// TwinCAT 3 PLC project TcAlarms
// Title: TwinCAT Alarm Handling Library
// Company: https://github.com/petr-suchy
// Author: Petr Suchý
// ProjectVersion: 0.0.1.0
// Description: TwinCAT library for alarm handling in PLC programs.
// ProgramVersion: 3.1.4024.0
// libraries:
//   Tc2_Standard, * (Beckhoff Automation GmbH)
//   Tc2_System, * (Beckhoff Automation GmbH)
//   Tc3_Module, * (Beckhoff Automation GmbH)
// project tree:
//   Alarms/DUTs/ E_AlarmSeverity.TcDUT, E_ArgType.TcDUT, ST_AlarmElement.TcDUT (not stored), ST_AlarmPageRow.TcDUT (not stored), ST_Arg.TcDUT (not stored)
//   Alarms/FBs/ FB_Alarm.TcPOU, FB_AlarmArg.TcPOU (not stored), FB_AlarmBase.TcPOU, FB_AlarmContext.TcPOU, FB_ArgStack.TcPOU, FB_RdArgStack.TcPOU, FB_SRAlarm.TcPOU (not stored), FB_SRAlarmArg.TcPOU, FB_VFormatStr.TcPOU, FB_WrArgStack.TcPOU
//   Alarms/FUNs/ A_BOOL.TcPOU (not stored), A_BYTE.TcPOU (not stored), A_DATE.TcPOU, A_DINT.TcPOU (not stored), A_DWORD.TcPOU (not stored), A_INT.TcPOU, A_LREAL.TcPOU (not stored), A_REAL.TcPOU, A_SINT.TcPOU (not stored), A_STRING.TcPOU (not stored), A_TIME.TcPOU, A_UDINT.TcPOU (not stored), A_UINT.TcPOU, A_USINT.TcPOU, A_WORD.TcPOU
//   Alarms/GVLs/ GVL_Alarms.TcGVL
//   Alarms/ITFs/ I_Alarm.TcIO, I_AlarmContext.TcIO, I_AlarmTextList.TcIO (not stored)
//   / ImagePool_Alarms.TcIPO (not stored), PlcTask.TcTTO
//   Memory/DUTs/ ST_SIZE.TcDUT
//   Memory/FUNs/ WORD_TO_SIZE.TcPOU, DINT_TO_SIZE.TcPOU, INT_TO_SIZE.TcPOU, F_MemCpy.TcPOU, F_MemSet.TcPOU, SINT_TO_SIZE.TcPOU, SIZE_TO_VALUE.TcPOU, UDINT_TO_SIZE.TcPOU, UINT_TO_SIZE.TcPOU, USINT_TO_SIZE.TcPOU, BYTE_TO_SIZE.TcPOU, DWORD_TO_SIZE.TcPOU
//   POUs/ MAIN.TcPOU
//   Version/ Global_Version.TcGVL
// real-time tasks:
//   TASK PlcTask: cycle T#10ms, priority 20, ADS port 350

CONFIGURATION TcAlarms
    RESOURCE PLC ON TwinCAT3
        TASK PlcTask(INTERVAL := T#10ms, PRIORITY := 20);
        PROGRAM MAIN WITH PlcTask : MAIN;
    END_RESOURCE
END_CONFIGURATION

// ---- Alarms/DUTs/E_AlarmSeverity.TcDUT
{attribute 'qualified_only'}
{attribute 'strict'}
{attribute 'to_string'}
TYPE E_AlarmSeverity :
(
	NoneAlarm := 0,
	InfoAlarm,
	WarningAlarm,
	ErrorAlarm
) BYTE := NoneAlarm;
END_TYPE

// ---- Alarms/DUTs/E_ArgType.TcDUT
{attribute 'qualified_only'}
{attribute 'strict'}
TYPE E_ArgType :
(
	VoidArg := 0,
	BoolArg,
	ByteArg,
	WordArg,
	DWordArg,
	SIntArg,
	USIntArg,
	IntArg,
	UIntArg,
	DIntArg,
	UDIntArg,
	RealArg,
	LRealArg,
	StringArg,
	TimeArg,
	DateArg
) BYTE := VoidArg;
END_TYPE

// ---- Memory/DUTs/ST_SIZE.TcDUT
TYPE ST_SIZE :
STRUCT
	nValue : UDINT;
END_STRUCT
END_TYPE

// ---- Alarms/GVLs/GVL_Alarms.TcGVL
VAR_GLOBAL CONSTANT
	ALARM_INVALID_CONTEXT_ID	: DINT := 0;
	ALARM_INVALID_INDEX			: DINT := -1;
	ALARM_ARG_STACK_SIZE		: DINT := 255;
	ALARM_TEXT_SIZE				: INT := 255;
END_VAR

// ---- Version/Global_Version.TcGVL
{attribute 'TcGenerated'}
{attribute 'no-analysis'}
{attribute 'linkalways'}
// This function has been automatically generated from the project information.
VAR_GLOBAL CONSTANT
	{attribute 'const_non_replaced'}
	stLibVersion_TwinCAT_Alarm_Handling_Library : ST_LibVersion := (iMajor := 0, iMinor := 0, iBuild := 1, iRevision := 0, nFlags := 0, sVersion := '0.0.1.0');
END_VAR

// ---- Alarms/ITFs/I_Alarm.TcIO
INTERFACE I_Alarm

PROPERTY AlarmId : DINT
GET
END_GET
END_PROPERTY

PROPERTY AlarmSeverity : E_AlarmSeverity
GET
END_GET
END_PROPERTY

PROPERTY ArgStackMemoryPointer : POINTER TO BYTE
GET
END_GET
END_PROPERTY

PROPERTY ArgStackMemorySize : DINT
GET
END_GET
END_PROPERTY

END_INTERFACE

// ---- Alarms/ITFs/I_AlarmContext.TcIO
INTERFACE I_AlarmContext

PROPERTY Acknowledge : BOOL
GET
END_GET
END_PROPERTY

METHOD AddNewAlarm : DINT
VAR_INPUT
	iAlarm : I_Alarm;
END_VAR
END_METHOD

METHOD EnableAcknowledge : BOOL
VAR_INPUT
	nAlarmContextId		: DINT;
	bCanByAcknowledged	: BOOL;
END_VAR
END_METHOD

PROPERTY IsAlarmBufferFull : BOOL
GET
END_GET
END_PROPERTY

METHOD RemoveAlarm : BOOL
VAR_INPUT
	nAlarmContextId : DINT;
END_VAR
END_METHOD

PROPERTY SelectedAlarmContextId : DINT
GET
END_GET
END_PROPERTY

END_INTERFACE

// ---- POUs/MAIN.TcPOU
PROGRAM MAIN
VAR
END_VAR

END_PROGRAM

// ---- Alarms/FBs/FB_Alarm.TcPOU
FUNCTION_BLOCK FB_Alarm EXTENDS FB_AlarmBase
VAR_INPUT
	bEnable				: BOOL;
END_VAR

bActive := bEnable;

SUPER^();

PROPERTY ArgStackMemoryPointer : POINTER TO BYTE
GET
ArgStackMemoryPointer := 0;
END_GET
END_PROPERTY

PROPERTY ArgStackMemorySize : DINT
GET
ArgStackMemorySize := 0;
END_GET
END_PROPERTY

METHOD PROTECTED  ClearArgStack
VAR_INPUT
END_VAR
// Do nothing
END_METHOD

METHOD PROTECTED CopyArgsToStack
VAR_INPUT
END_VAR
// Do nothing
END_METHOD

END_FUNCTION_BLOCK

// ---- Alarms/FBs/FB_AlarmBase.TcPOU
FUNCTION_BLOCK ABSTRACT FB_AlarmBase IMPLEMENTS I_Alarm
VAR_OUTPUT
	bActive				: BOOL;
END_VAR
VAR
	iAlarmContext		: I_AlarmContext;
	nAlarmContextId		: DINT := ALARM_INVALID_CONTEXT_ID;
	eAlarmSeverity		: E_AlarmSeverity;
	nAlarmId			: DINT;
	fbActiveRTrig		: R_TRIG;
	fbActiveFTrig		: F_TRIG;
END_VAR

fbActiveRTrig(CLK := bActive);
fbActiveFTrig(CLK := bActive);

IF fbActiveRTrig.Q THEN
	CopyArgsToStack();
END_IF

IF bActive AND nAlarmContextId = ALARM_INVALID_CONTEXT_ID AND NOT iAlarmContext.IsAlarmBufferFull THEN
	// Add this alarm to alarm context
	nAlarmContextId := iAlarmContext.AddNewAlarm(THIS^);
END_IF

IF fbActiveFTrig.Q THEN
	IF nAlarmContextId <> ALARM_INVALID_CONTEXT_ID THEN
		// Prepare argument stack for new arguments
		ClearArgStack();
		// Remove this alarm from alarm context
		iAlarmContext.RemoveAlarm(nAlarmContextId);
		nAlarmContextId := ALARM_INVALID_CONTEXT_ID;
	END_IF
END_IF

PROPERTY AlarmId : DINT
GET
AlarmId := nAlarmId;
END_GET
END_PROPERTY

PROPERTY AlarmSeverity : E_AlarmSeverity
GET
AlarmSeverity := eAlarmSeverity;
END_GET
END_PROPERTY

PROPERTY ABSTRACT ArgStackMemoryPointer : POINTER TO BYTE
GET
END_GET
END_PROPERTY

PROPERTY ABSTRACT ArgStackMemorySize : DINT
GET
END_GET
END_PROPERTY

METHOD PROTECTED ABSTRACT ClearArgStack
VAR_INPUT
END_VAR
END_METHOD

METHOD PROTECTED ABSTRACT CopyArgsToStack
VAR_INPUT
END_VAR
END_METHOD

METHOD FB_init : BOOL
VAR_INPUT
	bInitRetains		: BOOL; // if TRUE, the retain variables are initialized (warm start / cold start)
	bInCopyCode			: BOOL;  // if TRUE, the instance afterwards gets moved into the copy code (online change)
	iAlarmContext		: I_AlarmContext;
	eAlarmSeverity		: E_AlarmSeverity;
	nAlarmId			: DINT;
END_VAR
THIS^.iAlarmContext := iAlarmContext;
THIS^.eAlarmSeverity := eAlarmSeverity;
THIS^.nAlarmId := nAlarmId;
END_METHOD

END_FUNCTION_BLOCK

// ---- Alarms/FBs/FB_AlarmContext.TcPOU
FUNCTION_BLOCK FB_AlarmContext IMPLEMENTS I_AlarmContext
VAR_INPUT
	bEnable						: BOOL;
	bFirstAlarm					: BOOL;
	bLastAlarm					: BOOL;
	bPrevAlarm					: BOOL;
	bNextAlarm					: BOOL;
	bAcknowledge				: BOOL;
END_VAR
VAR_OUTPUT
	bActive						: BOOL;
	nNumOfDisplayedAlarms		: DINT;
END_VAR
VAR_IN_OUT
	aAlarmPage					: ARRAY[*] OF ST_AlarmPageRow;
	nSelectedAlarm				: INT;
END_VAR
VAR
	pAlarmArray					: POINTER TO ST_AlarmElement;
	nMaxNumOfAlarms				: DINT;
	iAlarmTextList				: I_AlarmTextList;
	nNumOfAlarms				: DINT;
	nNextContextId				: DINT := ALARM_INVALID_CONTEXT_ID + 1;
	nSelectedAlarmContextId		: DINT := ALARM_INVALID_CONTEXT_ID;
	fbEnableFTrig				: F_TRIG;
	fbFirstAlarmRTrig			: R_TRIG;
	fbLastAlarmRTrig			: R_TRIG;
	fbPrevAlarmRTrig			: R_TRIG;
	fbNextAlarmRTrig			: R_TRIG;
	fbVFormatStr				: FB_VFormatStr;
	// Index of the first alarm in the alarm array to be displayed
	nFirstAlarmToDisplay		: DINT;
	// Number of alarm selected in table
	nSelectedAlarm_				: DINT;
END_VAR
VAR_TEMP
	nPageLBound					: DINT;
	nPageUBound					: DINT;
	nPageSize					: DINT;
	nActualNumOfAlarms			: DINT;
	nSelectedAlarmOffset		: DINT;
	stCurrAlarm					: REFERENCE TO ST_AlarmElement;
	stCurrPageRow				: REFERENCE TO ST_AlarmPageRow;
	i							: DINT;
END_VAR

bActive := bEnable;
nSelectedAlarmContextId := ALARM_INVALID_CONTEXT_ID;

fbEnableFTrig(CLK := bEnable);

fbFirstAlarmRTrig(CLK := bFirstAlarm);
fbLastAlarmRTrig(CLK := bLastAlarm);
fbPrevAlarmRTrig(CLK := bPrevAlarm);
fbNextAlarmRTrig(CLK := bNextAlarm);

// The first index in the output array
nPageLBound := LOWER_BOUND(aAlarmPage, 1);
// The last index in the output array
nPageUBound := UPPER_BOUND(aAlarmPage, 1);
// Size of the output array
nPageSize := nPageUBound - nPageLBound + 1;

IF fbEnableFTrig.Q THEN
	// Reset FB output when enable is lost
	FOR i := nPageLBound TO nPageUBound DO
		ClearPageRow(i);
	END_FOR
	nNumOfDisplayedAlarms := 0;
END_IF

IF NOT bEnable THEN
	RETURN;
END_IF

// Get alarm number from FB input
nSelectedAlarm_ := nSelectedAlarm;

// Restrict index to the lower limit
nSelectedAlarm_ := MAX(nPageLBound, nSelectedAlarm_);
// Restrict index to the upper limit
nSelectedAlarm_ := MIN(nPageUBound, nSelectedAlarm_);

// Go to the first alarm
IF fbFirstAlarmRTrig.Q THEN
	nFirstAlarmToDisplay := 0;
	nSelectedAlarm_ := nPageLBound;
END_IF

// Go to the last alarm
IF fbLastAlarmRTrig.Q THEN
	nFirstAlarmToDisplay := (nNumOfAlarms / nPageSize) * nPageSize;
	nSelectedAlarm_ := MAX(nNumOfAlarms MOD nPageSize, 1);
END_IF

// Go to the previous alarm
IF fbPrevAlarmRTrig.Q THEN
	// Is the first alarm on the alarm page selected?
	IF nSelectedAlarm_ <= nPageLBound THEN
		// Move displayed alarms backward by one
		nFirstAlarmToDisplay := nFirstAlarmToDisplay - 1;
	ELSE
		// Select previous alarm
		nSelectedAlarm_ := nSelectedAlarm_ - 1;
	END_IF
END_IF

// Go to the next alarm
IF fbNextAlarmRTrig.Q THEN
	// Is the last alarm on the alarm page selected?
	IF nSelectedAlarm_ >= nPageUBound THEN
		IF nNumOfAlarms > nPageSize THEN
			// Move displayed alarms forward by one
			nFirstAlarmToDisplay := nFirstAlarmToDisplay + 1;
		END_IF
	ELSE
		// Select next alarm
		nSelectedAlarm_ := nSelectedAlarm_ + 1;
	END_IF
END_IF

// Return selected alarm back to the FB output
nSelectedAlarm := DINT_TO_INT(nSelectedAlarm_);

// Restrict alarm index to the upper limit
nFirstAlarmToDisplay := MIN(nFirstAlarmToDisplay, nNumOfAlarms - 1);
// Restrict alarm index to the lower limit
nFirstAlarmToDisplay := MAX(nFirstAlarmToDisplay, 0);

// Actual number of alarms that can be displayed
nActualNumOfAlarms := nNumOfAlarms - nFirstAlarmToDisplay;
// Number of alarms to be displayed
nNumOfDisplayedAlarms := MIN(nPageSize, nActualNumOfAlarms);

FOR i := 0 TO nNumOfDisplayedAlarms - 1 DO
	
	stCurrAlarm REF= pAlarmArray[nFirstAlarmToDisplay + i];
	stCurrPageRow REF= aAlarmPage[nPageLBound + i];

	// Convert alarm severity to string
	stCurrPageRow.sAlarmSeverity := TO_STRING(stCurrAlarm.eAlarmSeverity);
	// Convert alarm id to string
	stCurrPageRow.sAlarmId := DINT_TO_STRING(stCurrAlarm.nAlarmId);	
	// Format alarm text using the argument stack
	fbVFormatStr(
		sFormat := iAlarmTextList.GetAlarmText(stCurrAlarm.nAlarmId),
		pArgStack := ADR(stCurrAlarm.aArgStack), 
		nStackSize := SIZEOF(stCurrAlarm.aArgStack),
		sOutput => stCurrPageRow.sAlarmText
	);
	// Convert Ack flag to string
	IF stCurrAlarm.bCanByAcknowledged THEN
		stCurrPageRow.sCanByAcknowledged := '!';
	ELSE
		stCurrPageRow.sCanByAcknowledged := '';
	END_IF
END_FOR

// Clear the rest of the output array
FOR i := nPageLBound + nNumOfDisplayedAlarms TO nPageUBound DO
	ClearPageRow(i);
END_FOR

// Get context id of selected alarm
IF nPageLBound <= nSelectedAlarm_ AND nSelectedAlarm_ <= nPageUBound THEN
	nSelectedAlarmOffset := nSelectedAlarm_ - nPageLBound;
	IF nSelectedAlarmOffset < nNumOfDisplayedAlarms THEN
		nSelectedAlarmContextId := pAlarmArray[nFirstAlarmToDisplay + nSelectedAlarmOffset].nAlarmContextId;
	END_IF
END_IF

PROPERTY Acknowledge : BOOL
GET
Acknowledge := bAcknowledge;
END_GET
END_PROPERTY

METHOD PUBLIC AddNewAlarm : DINT
VAR_INPUT
	iAlarm : I_Alarm;
END_VAR
VAR
	i : DINT;
END_VAR
AddNewAlarm := ALARM_INVALID_CONTEXT_ID;

IF NOT IsAlarmBufferFull THEN

	// Make space for a new alarm by shifting array elements to right
	FOR i := 1 TO nNumOfAlarms DO
		pAlarmArray[nNumOfAlarms - i + 1] := pAlarmArray[nNumOfAlarms - i];
	END_FOR
	
	pAlarmArray[0].nAlarmContextId := nNextContextId;
	pAlarmArray[0].eAlarmSeverity := iAlarm.AlarmSeverity; 
	pAlarmArray[0].nAlarmId := iAlarm.AlarmId;
	pAlarmArray[0].bCanByAcknowledged := FALSE;
	
	IF iAlarm.ArgStackMemoryPointer <> 0 AND iAlarm.ArgStackMemorySize > 0 THEN
		F_MemCpy(
			pDestAddr:= ADR(pAlarmArray[0].aArgStack),
			stDestSize:= UDINT_TO_SIZE(SIZEOF(pAlarmArray[0].aArgStack)),
			pSrcAddr:= iAlarm.ArgStackMemoryPointer,
			stSrcSize:= DINT_TO_SIZE(iAlarm.ArgStackMemorySize));
	END_IF

	nNextContextId := nNextContextId + 1;
	
	// Prevent context id overflow
	IF nNextContextId <= ALARM_INVALID_CONTEXT_ID THEN
		nNextContextId := ALARM_INVALID_CONTEXT_ID + 1;
	END_IF
	
	nNumOfAlarms := nNumOfAlarms + 1;

	AddNewAlarm := pAlarmArray[0].nAlarmContextId;
END_IF
END_METHOD

METHOD PRIVATE ClearPageRow
VAR_INPUT
	nRowIdx : DINT;
END_VAR
aAlarmPage[nRowIdx].sAlarmSeverity := TO_STRING(E_AlarmSeverity.NoneAlarm);
aAlarmPage[nRowIdx].sAlarmId := '';
aAlarmPage[nRowIdx].sAlarmText := '';
aAlarmPage[nRowIdx].sCanByAcknowledged := '';
END_METHOD

METHOD PUBLIC EnableAcknowledge : BOOL
VAR_INPUT
	nAlarmContextId		: DINT;
	bCanByAcknowledged	: BOOL;
END_VAR
VAR
	nArrayIndex			: DINT;
END_VAR
EnableAcknowledge := FALSE;
nArrayIndex := GetArrayIndexByContextId(nAlarmContextId);

IF nArrayIndex <> ALARM_INVALID_INDEX THEN
	pAlarmArray[nArrayIndex].bCanByAcknowledged := bCanByAcknowledged;
	EnableAcknowledge := TRUE;
END_IF
END_METHOD

METHOD FB_init : BOOL
VAR_INPUT
	bInitRetains			: BOOL;								// if TRUE, the retain variables are initialized (warm start / cold start)
	bInCopyCode				: BOOL;								// if TRUE, the instance afterwards gets moved into the copy code (online change)
	pAlarmArray				: POINTER TO ST_AlarmElement;
	nMaxNumOfAlarms			: DINT;
	iAlarmTextList			: I_AlarmTextList;
END_VAR
THIS^.pAlarmArray := pAlarmArray;
THIS^.nMaxNumOfAlarms := nMaxNumOfAlarms;
THIS^.iAlarmTextList := iAlarmTextList;
END_METHOD

METHOD PRIVATE GetArrayIndexByContextId : DINT
VAR_INPUT
	nAlarmContextId : DINT;
END_VAR
VAR
	i : DINT;
END_VAR
GetArrayIndexByContextId := ALARM_INVALID_INDEX;

IF nAlarmContextId <> ALARM_INVALID_CONTEXT_ID THEN
	FOR i := 0 TO nNumOfAlarms - 1 DO
		IF pAlarmArray[i].nAlarmContextId = nAlarmContextId THEN
			GetArrayIndexByContextId := i;
			RETURN;
		END_IF
	END_FOR
END_IF
END_METHOD

PROPERTY PUBLIC IsAlarmBufferFull : BOOL
GET
IsAlarmBufferFull := nNumOfAlarms >= nMaxNumOfAlarms;
END_GET
END_PROPERTY

METHOD PUBLIC RemoveAlarm : BOOL
VAR_INPUT
	nAlarmContextId		: DINT;
END_VAR
VAR
	nArrayIndex			: DINT;
	i					: DINT;
END_VAR
RemoveAlarm := FALSE;
nArrayIndex := GetArrayIndexByContextId(nAlarmContextId);

IF nArrayIndex > ALARM_INVALID_INDEX AND nArrayIndex < nNumOfAlarms THEN

	// Remove element from array by shifting array elements to left
	FOR i := nArrayIndex TO nNumOfAlarms - 2 DO
		pAlarmArray[i] := pAlarmArray[i + 1];
	END_FOR
	nNumOfAlarms := nNumOfAlarms - 1;
	
	// Reinitialise element at the end of array freed by shifting
	pAlarmArray[nNumOfAlarms].nAlarmContextId := ALARM_INVALID_CONTEXT_ID;
	pAlarmArray[nNumOfAlarms].nAlarmId := 0;
	pAlarmArray[nNumOfAlarms].bCanByAcknowledged := FALSE;
	
	F_MemSet(
		pDestAddr:= ADR(pAlarmArray[nNumOfAlarms].aArgStack),
		nWithChar:= 0,
		stDestSize:= UDINT_TO_SIZE(SIZEOF(pAlarmArray[nNumOfAlarms].aArgStack)));

	RemoveAlarm := TRUE;
END_IF
END_METHOD

PROPERTY PUBLIC SelectedAlarmContextId : DINT
GET
SelectedAlarmContextId := nSelectedAlarmContextId;
END_GET
END_PROPERTY

END_FUNCTION_BLOCK

// ---- Alarms/FBs/FB_VFormatStr.TcPOU
FUNCTION_BLOCK FB_VFormatStr
VAR_INPUT
	sFormat			: STRING(ALARM_TEXT_SIZE);
	pArgStack		: POINTER TO BYTE;
	nStackSize		: DINT;
END_VAR
VAR_OUTPUT
	sOutput			: STRING(ALARM_TEXT_SIZE);
END_VAR
VAR
	fbRdArgStack		: FB_RdArgStack(0, 0);
	nFormatLength		: INT;
	nCurrFormatIndex	: INT;
	nCurrOutputIndex	: INT;
	i					: INT;
	c					: BYTE;
END_VAR
VAR CONSTANT
	SPEC_CHAR	: BYTE := 37;	// '%'
	SPEC_D		: BYTE := 100;	// '%d'
	SPEC_F		: BYTE := 102;	// '%f'
	SPEC_S		: BYTE := 115;	// '%s'
	SPEC_TIME	: BYTE := 84;	// %T
	SPEC_DATE	: BYTE := 68;	// %D
END_VAR

fbRdArgStack.SetMemory(pArgStack, nStackSize);

// Zero output string
F_MemSet(
	pDestAddr:= ADR(sOutput),
	nWithChar:= 0,
	stDestSize:= UDINT_TO_SIZE(SIZEOF(sOutput)));

// Get format string length
nFormatLength := LEN(sFormat);

nCurrFormatIndex := 0;
nCurrOutputIndex := 0;

WHILE NOT AtFmtEnd DO
	
	c := FmtChar;
	NextFmtChar();
	
	IF c = SPEC_CHAR THEN
		
		IF AtFmtEnd THEN
			PutChar(c);
			EXIT;
		END_IF
		
		c := FmtChar;
		NextFmtChar();
	
		CASE c OF
			SPEC_D:
				IF fbRdArgStack.IsIntArg THEN
					PutStr(DINT_TO_STRING(fbRdArgStack.GetIntArg()));
				ELSIF fbRdArgStack.IsUIntArg THEN
					PutStr(UDINT_TO_STRING(fbRdArgStack.GetUIntArg()));
				ELSE
					PutStr('???');
				END_IF
				fbRdArgStack.NextArg();
			SPEC_F:
				IF fbRdArgStack.IsFloatArg THEN
					PutStr(LREAL_TO_STRING(fbRdArgStack.GetFloatArg()));
				ELSE
					PutStr('???');
				END_IF
				fbRdArgStack.NextArg();
			SPEC_S:
				IF fbRdArgStack.IsString THEN
					PutStr(fbRdArgStack.GetStringArg());
				ELSE
					PutStr('???');
				END_IF
			SPEC_TIME:
				IF fbRdArgStack.IsTime THEN
					PutStr(TIME_TO_STRING(fbRdArgStack.GetTimeArg()));
				ELSE
					PutStr('???');
				END_IF
			SPEC_DATE:
				IF fbRdArgStack.IsDate THEN
					PutStr(DATE_TO_STRING(fbRdArgStack.GetDateArg()));
				ELSE
					PutStr('???');
				END_IF			
		ELSE
			IF c = SPEC_CHAR THEN // %% escape sequence?
				PutChar(c);
			ELSE
				PutChar(SPEC_CHAR);
				PutChar(c);
			END_IF
		END_CASE
	ELSE
		PutChar(c);
	END_IF
END_WHILE

PROPERTY PRIVATE AtFmtEnd : BOOL
GET
AtFmtEnd := nCurrFormatIndex >= nFormatLength;
END_GET
END_PROPERTY

PROPERTY PRIVATE FmtChar : BYTE
GET
FmtChar := sFormat[nCurrFormatIndex];
END_GET
END_PROPERTY

METHOD PRIVATE NextFmtChar
VAR_INPUT
END_VAR
IF nCurrFormatIndex < nFormatLength THEN
	nCurrFormatIndex := nCurrFormatIndex + 1;
END_IF
END_METHOD

METHOD PRIVATE PutChar
VAR_INPUT
	nOutChar : BYTE;
END_VAR
IF nCurrOutputIndex < ALARM_TEXT_SIZE THEN
	sOutput[nCurrOutputIndex] := nOutChar;
	nCurrOutputIndex := nCurrOutputIndex + 1;
END_IF
END_METHOD

METHOD PRIVATE PutStr
VAR_INPUT
	sOutStr : STRING(ALARM_TEXT_SIZE);
END_VAR
VAR
	nOutStrLen	: INT;
	i			: INT;
END_VAR
nOutStrLen := LEN(sOutStr);

i := 0;
WHILE i < nOutStrLen AND nCurrOutputIndex < ALARM_TEXT_SIZE DO
	sOutput[nCurrOutputIndex] := sOutStr[i];
	i := i + 1;
	nCurrOutputIndex := nCurrOutputIndex + 1;
END_WHILE
END_METHOD

END_FUNCTION_BLOCK

// ---- Alarms/FBs/FB_RdArgStack.TcPOU
FUNCTION_BLOCK FB_RdArgStack EXTENDS FB_ArgStack

PROPERTY PUBLIC AtEnd : BOOL
GET
AtEnd := AtEndOfMemory;
END_GET
END_PROPERTY

METHOD PUBLIC GetDateArg : DATE
VAR
	pDate : POINTER TO DATE;
END_VAR
IF ArgDataAvailableSize < ArgSize THEN
	RETURN;
END_IF

IF IsDate AND ArgSize = SIZEOF(pDate^) THEN
	pDate := ArgDataPointer;
	GetDateArg := pDate^;
END_IF
END_METHOD

METHOD GetFloatArg : LREAL
VAR
	pReal		: POINTER TO REAL;
	pLReal		: POINTER TO LREAL;
END_VAR

IF ArgDataAvailableSize < ArgSize THEN
	RETURN;
END_IF

CASE ArgType OF
	E_ArgType.RealArg:
		IF ArgSize = SIZEOF(pReal^) THEN
			pReal := ArgDataPointer;
			GetFloatArg := pReal^;
		END_IF

	E_ArgType.LRealArg:
		IF ArgSize = SIZEOF(pLReal^) THEN
			pLReal := ArgDataPointer;
			GetFloatArg := pLReal^;
		END_IF

END_CASE
END_METHOD

METHOD PUBLIC GetIntArg : DINT
VAR
	pSInt		: POINTER TO SINT;
	pInt		: POINTER TO INT;
	pDInt		: POINTER TO DINT;
END_VAR

IF ArgDataAvailableSize < ArgSize THEN
	RETURN;
END_IF

CASE ArgType OF
	E_ArgType.SIntArg:
		IF ArgSize = SIZEOF(pSInt^) THEN
			pSInt := ArgDataPointer;
			GetIntArg := pSInt^;
		END_IF

	E_ArgType.IntArg:
		IF ArgSize = SIZEOF(pInt^) THEN
			pInt := ArgDataPointer;
			GetIntArg := pInt^;
		END_IF
		
	E_ArgType.DIntArg:
		IF ArgSize = SIZEOF(pDInt^) THEN
			pDInt := ArgDataPointer;
			GetIntArg := pDInt^;
		END_IF

END_CASE
END_METHOD

METHOD PUBLIC GetStringArg : STRING
VAR
	nStrLen		: INT;
	nMaxOutLen	: INT;
	i			: INT;
	j			: DINT;
END_VAR
IF ArgDataAvailableSize < ArgSize THEN
	RETURN;
END_IF

nStrLen := ArgSize;
nMaxOutLen := UDINT_TO_INT(SIZEOF(GetStringArg));

i := 0;
j := ArgDataOffset;

WHILE i < nStrLen AND i < nMaxOutLen DO
	GetStringArg[i] := pStackMemory[j];
	i := i + 1;
	j := j + 1;
END_WHILE

GetStringArg[i] := 0;
END_METHOD

METHOD PUBLIC GetTimeArg : TIME
VAR
	pTime : POINTER TO TIME;
END_VAR
IF ArgDataAvailableSize < ArgSize THEN
	RETURN;
END_IF

IF IsTime AND ArgSize = SIZEOF(pTime^) THEN
	pTime := ArgDataPointer;
	GetTimeArg := pTime^;
END_IF
END_METHOD

METHOD PUBLIC GetUIntArg : UDINT
VAR
	pByte		: POINTER TO BYTE;
	pWord		: POINTER TO WORD;
	pDWord		: POINTER TO DWORD;
	pUSInt		: POINTER TO USINT;
	pUInt		: POINTER TO UINT;
	pUDInt		: POINTER TO UDINT;
END_VAR

IF ArgDataAvailableSize < ArgSize THEN
	RETURN;
END_IF

CASE ArgType OF
	E_ArgType.ByteArg:
		IF ArgSize = SIZEOF(pByte^) THEN
			pByte := ArgDataPointer;
			GetUIntArg := pByte^;
		END_IF
		
	E_ArgType.WordArg:
		IF ArgSize = SIZEOF(pWord^) THEN
			pWord := ArgDataPointer;
			GetUIntArg := pWord^;
		END_IF
		
	E_ArgType.DWordArg:
		IF ArgSize = SIZEOF(pDWord^) THEN
			pDWord := ArgDataPointer;
			GetUIntArg := pDWord^;
		END_IF
		
	E_ArgType.USIntArg:
		IF ArgSize = SIZEOF(pUSInt^) THEN
			pUSInt := ArgDataPointer;
			GetUIntArg := pUSInt^;
		END_IF

	E_ArgType.UIntArg:
		IF ArgSize = SIZEOF(pUInt^) THEN
			pUInt := ArgDataPointer;
			GetUIntArg := pUInt^;
		END_IF

	E_ArgType.UDIntArg:
		IF ArgSize = SIZEOF(pUDInt^) THEN
			pUDInt := ArgDataPointer;
			GetUIntArg := pUDInt^;
		END_IF
		
END_CASE
END_METHOD

PROPERTY PUBLIC IsDate : BOOL
GET
IsDate := ArgType = E_ArgType.DateArg;
END_GET
END_PROPERTY

PROPERTY PUBLIC IsFloatArg : BOOL
GET
IsFloatArg := ArgType = E_ArgType.RealArg OR
	ArgType = E_ArgType.LRealArg;
END_GET
END_PROPERTY

PROPERTY PUBLIC IsIntArg : BOOL
GET
IsIntArg := ArgType = E_ArgType.SIntArg OR
	ArgType = E_ArgType.IntArg OR
	ArgType = E_ArgType.DIntArg;
END_GET
END_PROPERTY

PROPERTY PUBLIC IsString : BOOL
GET
IsString := ArgType = E_ArgType.StringArg;
END_GET
END_PROPERTY

PROPERTY PUBLIC IsTime : BOOL
GET
IsTime := ArgType = E_ArgType.TimeArg;
END_GET
END_PROPERTY

PROPERTY PUBLIC IsUIntArg : BOOL
GET
IsUIntArg := ArgType = E_ArgType.USIntArg OR
	ArgType = E_ArgType.UIntArg OR
	ArgType = E_ArgType.UDIntArg;
END_GET
END_PROPERTY

METHOD PUBLIC NextArg
VAR_INPUT
END_VAR
nCurrOfsetInStack := MIN(nCurrOfsetInStack + ARG_HEADER_SIZE + ArgSize, nStackMemorySize);
END_METHOD

METHOD PUBLIC Reset : DINT
VAR_INPUT
END_VAR
nCurrOfsetInStack := 0;
END_METHOD

END_FUNCTION_BLOCK

// ---- Alarms/FBs/FB_ArgStack.TcPOU
FUNCTION_BLOCK FB_ArgStack
VAR_INPUT
END_VAR
VAR_OUTPUT
END_VAR
VAR
	pStackMemory			: POINTER TO BYTE;
	nStackMemorySize		: DINT;
	nCurrOfsetInStack		: DINT;
END_VAR
VAR CONSTANT
	ARG_HEADER_SIZE			: DINT := 2;
END_VAR

PROPERTY PROTECTED ArgDataAvailableSize : DINT
GET
ArgDataAvailableSize := MAX(0, RemainingMemorySize - ARG_HEADER_SIZE);
END_GET
END_PROPERTY

PROPERTY PROTECTED ArgDataOffset : DINT
GET
ArgDataOffset := nCurrOfsetInStack + ARG_HEADER_SIZE;
END_GET
END_PROPERTY

PROPERTY PUBLIC ArgDataPointer : POINTER TO BYTE
GET
ArgDataPointer := ADR(pStackMemory[ArgDataOffset]);
END_GET
END_PROPERTY

PROPERTY PROTECTED ArgSize : BYTE
GET
ArgSize := pStackMemory[nCurrOfsetInStack + 1];
END_GET
SET
pStackMemory[nCurrOfsetInStack + 1] := ArgSize;
END_SET
END_PROPERTY

PROPERTY PROTECTED ArgType : BYTE
GET
ArgType := pStackMemory[nCurrOfsetInStack];
END_GET
SET
pStackMemory[nCurrOfsetInStack] := ArgType;
END_SET
END_PROPERTY

PROPERTY PROTECTED AtEndOfMemory : BOOL
GET
AtEndOfMemory := RemainingMemorySize < ARG_HEADER_SIZE;
END_GET
END_PROPERTY

METHOD PUBLIC Clear
nCurrOfsetInStack := 0;

IF nStackMemorySize > 0 THEN
	// Zero stack memory
	F_MemSet(
		pDestAddr:= pStackMemory,
		nWithChar:= 0,
		stDestSize:= DINT_TO_SIZE(nStackMemorySize));
END_IF
END_METHOD

METHOD FB_init : BOOL
VAR_INPUT
	bInitRetains		: BOOL; // if TRUE, the retain variables are initialized (warm start / cold start)
	bInCopyCode			: BOOL;  // if TRUE, the instance afterwards gets moved into the copy code (online change)
	pStackMemory		: POINTER TO BYTE;
	nStackMemorySize	: DINT;
END_VAR
SetMemory(pStackMemory, nStackMemorySize);
END_METHOD

PROPERTY PUBLIC MemoryPointer : POINTER TO BYTE
GET
MemoryPointer := pStackMemory;
END_GET
END_PROPERTY

PROPERTY PUBLIC MemorySize : DINT
GET
MemorySize := nStackMemorySize;
END_GET
END_PROPERTY

PROPERTY PROTECTED RemainingMemorySize : DINT
GET
RemainingMemorySize := nStackMemorySize - nCurrOfsetInStack;
END_GET
END_PROPERTY

METHOD PUBLIC SetMemory
VAR_INPUT
	pStackMemory		: POINTER TO BYTE;
	nStackMemorySize	: DINT;
END_VAR
THIS^.pStackMemory := pStackMemory;

IF THIS^.pStackMemory <> 0 THEN
	THIS^.nStackMemorySize := nStackMemorySize;
ELSE
	THIS^.nStackMemorySize := 0;
END_IF

THIS^.nCurrOfsetInStack := 0;
END_METHOD

PROPERTY PUBLIC UsedMemorySize : DINT
GET
UsedMemorySize := nCurrOfsetInStack;
END_GET
END_PROPERTY

END_FUNCTION_BLOCK

// ---- Memory/FUNs/F_MemSet.TcPOU
FUNCTION F_MemSet : DINT
VAR_INPUT
	pDestAddr			: POINTER TO BYTE;
	nWithChar			: BYTE;
	stDestSize			: ST_SIZE;
END_VAR
VAR
	nNumOfBytesToFill	: UDINT;
END_VAR

nNumOfBytesToFill := SIZE_TO_VALUE(stDestSize);

{IF defined (pou: MEMUtils.MemSet)}
    // CODESYS implementation
	MEMUtils.MemSet(
		pbyBuffer := pDestAddr,
		byValue := nWithChar,
		dwSize := nNumOfBytesToFill);
{ELSE}
	// TwinCAT implementation
	MEMSET(
		destAddr:= pDestAddr,
		fillByte:= nWithChar,
		n:= nNumOfBytesToFill);
{END_IF}

F_MemSet := UDINT_TO_DINT(nNumOfBytesToFill);

END_FUNCTION

// ---- Memory/FUNs/SIZE_TO_VALUE.TcPOU
FUNCTION SIZE_TO_VALUE : UDINT
VAR_INPUT
	stSize : ST_SIZE;
END_VAR

SIZE_TO_VALUE := stSize.nValue;

END_FUNCTION

// ---- Memory/FUNs/DINT_TO_SIZE.TcPOU
FUNCTION DINT_TO_SIZE : ST_SIZE
VAR_INPUT
	nValue : DINT;
END_VAR

DINT_TO_SIZE.nValue := DINT_TO_UDINT(MAX(0, nValue));

END_FUNCTION

// ---- Memory/FUNs/UDINT_TO_SIZE.TcPOU
FUNCTION UDINT_TO_SIZE : ST_SIZE
VAR_INPUT
	nValue : UDINT;
END_VAR

UDINT_TO_SIZE.nValue := nValue;

END_FUNCTION

// ---- Memory/FUNs/F_MemCpy.TcPOU
FUNCTION F_MemCpy : DINT
VAR_INPUT
	pDestAddr	: POINTER TO BYTE;
	stDestSize	: ST_SIZE;
	pSrcAddr	: POINTER TO BYTE;
	stSrcSize	: ST_SIZE;
END_VAR
VAR
	nNumOfBytesToCopy : UDINT;
END_VAR

nNumOfBytesToCopy := MIN(SIZE_TO_VALUE(stDestSize), SIZE_TO_VALUE(stSrcSize));

{IF defined (pou: MEMUtils.MemCpy)}
    // CODESYS implementation
	MEMUtils.MemCpy(
		pbyDest := pDestAddr,
		pbySrc := pSrcAddr,
		dwSize := nNumOfBytesToCopy);
{ELSE}
	// TwinCAT implementation
	MEMCPY(
		destAddr:= pDestAddr,
		srcAddr:= pSrcAddr,
		n:= nNumOfBytesToCopy);
{END_IF}

F_MemCpy := UDINT_TO_DINT(nNumOfBytesToCopy);

END_FUNCTION

// ---- Alarms/FBs/FB_SRAlarmArg.TcPOU
FUNCTION_BLOCK FB_SRAlarmArg EXTENDS FB_SRAlarm
VAR_INPUT
    arg1		: ST_Arg;
    arg2		: ST_Arg;
	arg3		: ST_Arg;
	arg4		: ST_Arg;
	arg5		: ST_Arg;
END_VAR
VAR
	aArgStack			: ARRAY[1..ALARM_ARG_STACK_SIZE] OF BYTE;
	fbWritableArgStack	: FB_WrArgStack(ADR(aArgStack), ALARM_ARG_STACK_SIZE);
END_VAR

SUPER^();

PROPERTY ArgStackMemoryPointer : POINTER TO BYTE
GET
ArgStackMemoryPointer := fbWritableArgStack.MemoryPointer;
END_GET
END_PROPERTY

PROPERTY ArgStackMemorySize : DINT
GET
ArgStackMemorySize := fbWritableArgStack.MemorySize;
END_GET
END_PROPERTY

METHOD PROTECTED  ClearArgStack
VAR_INPUT
END_VAR
fbWritableArgStack.Clear();
END_METHOD

METHOD PROTECTED CopyArgsToStack
VAR_INPUT
END_VAR
fbWritableArgStack.AddArg(arg1);
fbWritableArgStack.AddArg(arg2);
fbWritableArgStack.AddArg(arg3);
fbWritableArgStack.AddArg(arg4);
fbWritableArgStack.AddArg(arg5);
END_METHOD

END_FUNCTION_BLOCK

// ---- Alarms/FBs/FB_WrArgStack.TcPOU
FUNCTION_BLOCK FB_WrArgStack EXTENDS FB_ArgStack

METHOD PUBLIC AddArg : DINT
VAR_INPUT
	stArg : ST_Arg;
END_VAR
VAR
	eArgType				: E_ArgType;
	nArgSize				: BYTE;
END_VAR
// Return zero if there is not enough space to write argument
AddArg := 0;

// Is there enough space to write the entire argument?
IF ARG_HEADER_SIZE + stArg.nSize <= RemainingMemorySize THEN
	nArgSize := stArg.nSize;
ELSE
	// Can a string argument be truncated?
	IF stArg.eType = E_ArgType.StringArg AND RemainingMemorySize >= ARG_HEADER_SIZE THEN
		nArgSize := DINT_TO_BYTE(RemainingMemorySize - ARG_HEADER_SIZE);
	ELSE
		RETURN;
	END_IF
END_IF

// Is a pointer to the argument data provided?
IF stArg.pData <> 0 THEN
	eArgType := stArg.eType;
ELSE
	// Write void argument to the stack memory
	eArgType := E_ArgType.VoidArg;
	nArgSize := 0;
END_IF

// Write argument type and its size to the stack memory
ArgType := eArgType;
ArgSize := nArgSize;

// Write argument data to the stack memory
F_MemCpy(
	pDestAddr:= ArgDataPointer,
	stDestSize:= DINT_TO_SIZE(MemorySize - ArgDataOffset),
	pSrcAddr:= stArg.pData,
	stSrcSize:= BYTE_TO_SIZE(stArg.nSize));
	
// Add the header length and argument size to the current position in the stack memory
nCurrOfsetInStack := nCurrOfsetInStack + ARG_HEADER_SIZE + nArgSize;

// Return number of bytes written to the stack memory
AddArg := ARG_HEADER_SIZE + nArgSize;
END_METHOD

PROPERTY PUBLIC BytesWritten : DINT
GET
BytesWritten := UsedMemorySize;
END_GET
END_PROPERTY

PROPERTY IsFull : BOOL
GET
IsFull := AtEndOfMemory;
END_GET
END_PROPERTY

END_FUNCTION_BLOCK

// ---- Memory/FUNs/BYTE_TO_SIZE.TcPOU
FUNCTION BYTE_TO_SIZE : ST_SIZE
VAR_INPUT
	nValue : BYTE;
END_VAR

BYTE_TO_SIZE.nValue := nValue;

END_FUNCTION

// ---- Alarms/FUNs/A_DATE.TcPOU
FUNCTION A_DATE : ST_Arg
VAR_INPUT
	obj	: REFERENCE TO DATE;
END_VAR

IF __ISVALIDREF(obj) THEN
	A_DATE.eType := E_ArgType.DateArg;
	A_DATE.pData := ADR(obj);
	A_DATE.nSize := SIZEOF(DATE);
END_IF

END_FUNCTION

// ---- Alarms/FUNs/A_INT.TcPOU
FUNCTION A_INT : ST_Arg
VAR_INPUT
	nNumber	: REFERENCE TO INT;
END_VAR

IF __ISVALIDREF(nNumber) THEN
	A_INT.eType := E_ArgType.IntArg;
	A_INT.pData := ADR(nNumber);
	A_INT.nSize := SIZEOF(INT);
END_IF

END_FUNCTION

// ---- Alarms/FUNs/A_REAL.TcPOU
FUNCTION A_REAL : ST_Arg
VAR_INPUT
	fNumber	: REFERENCE TO REAL;
END_VAR

IF __ISVALIDREF(fNumber) THEN
	A_REAL.eType := E_ArgType.RealArg;
	A_REAL.pData := ADR(fNumber);
	A_REAL.nSize := SIZEOF(REAL);
END_IF

END_FUNCTION

// ---- Alarms/FUNs/A_TIME.TcPOU
FUNCTION A_TIME : ST_Arg
VAR_INPUT
	obj	: REFERENCE TO TIME;
END_VAR

IF __ISVALIDREF(obj) THEN
	A_TIME.eType := E_ArgType.TimeArg;
	A_TIME.pData := ADR(obj);
	A_TIME.nSize := SIZEOF(TIME);
END_IF

END_FUNCTION

// ---- Alarms/FUNs/A_UINT.TcPOU
FUNCTION A_UINT : ST_Arg
VAR_INPUT
	nNumber	: REFERENCE TO UINT;
END_VAR

IF __ISVALIDREF(nNumber) THEN
	A_UINT.eType := E_ArgType.UIntArg;
	A_UINT.pData := ADR(nNumber);
	A_UINT.nSize := SIZEOF(UINT);
END_IF

END_FUNCTION

// ---- Alarms/FUNs/A_USINT.TcPOU
FUNCTION A_USINT : ST_Arg
VAR_INPUT
	nNumber	: REFERENCE TO USINT;
END_VAR

IF __ISVALIDREF(nNumber) THEN
	A_USINT.eType := E_ArgType.USIntArg;
	A_USINT.pData := ADR(nNumber);
	A_USINT.nSize := SIZEOF(USINT);
END_IF

END_FUNCTION

// ---- Alarms/FUNs/A_WORD.TcPOU
FUNCTION A_WORD : ST_Arg
VAR_INPUT
	nNumber	: REFERENCE TO WORD;
END_VAR

IF __ISVALIDREF(nNumber) THEN
	A_WORD.eType := E_ArgType.WordArg;
	A_WORD.pData := ADR(nNumber);
	A_WORD.nSize := SIZEOF(WORD);
END_IF

END_FUNCTION

// ---- Memory/FUNs/WORD_TO_SIZE.TcPOU
FUNCTION WORD_TO_SIZE : ST_SIZE
VAR_INPUT
	nValue : WORD;
END_VAR

WORD_TO_SIZE.nValue := nValue;

END_FUNCTION

// ---- Memory/FUNs/INT_TO_SIZE.TcPOU
FUNCTION INT_TO_SIZE : ST_SIZE
VAR_INPUT
	nValue : INT;
END_VAR

INT_TO_SIZE.nValue := INT_TO_UDINT(MAX(0, nValue));

END_FUNCTION

// ---- Memory/FUNs/SINT_TO_SIZE.TcPOU
FUNCTION SINT_TO_SIZE : ST_SIZE
VAR_INPUT
	nValue : SINT;
END_VAR

SINT_TO_SIZE.nValue := SINT_TO_UDINT(MAX(0, nValue));

END_FUNCTION

// ---- Memory/FUNs/UINT_TO_SIZE.TcPOU
FUNCTION UINT_TO_SIZE : ST_SIZE
VAR_INPUT
	nValue : UINT;
END_VAR

UINT_TO_SIZE.nValue := nValue;

END_FUNCTION

// ---- Memory/FUNs/USINT_TO_SIZE.TcPOU
FUNCTION USINT_TO_SIZE : ST_SIZE
VAR_INPUT
	nValue : USINT;
END_VAR

USINT_TO_SIZE.nValue := nValue;

END_FUNCTION

// ---- Memory/FUNs/DWORD_TO_SIZE.TcPOU
FUNCTION DWORD_TO_SIZE : ST_SIZE
VAR_INPUT
	nValue : DWORD;
END_VAR

DWORD_TO_SIZE.nValue := nValue;

END_FUNCTION
